PROGRAM PRG_ReadInputs
VAR
END_VAR

// -----------------------------------------------------------------------------
// OPERATOR CONTROLS
// -----------------------------------------------------------------------------
GVL_MASTER.stInputs.bStartButton                       := GVL_IO.stInputs.bStartButton;
GVL_MASTER.stInputs.bStopButton                        := GVL_IO.stInputs.bStopButton;
GVL_MASTER.stInputs.bResetButton                       := GVL_IO.stInputs.bResetButton;
GVL_MASTER.stInputs.bTwoHandsSafe                      := GVL_IO.stInputs.bTwoHandsSafe;

// -----------------------------------------------------------------------------
// PHYSICAL SAFETY DIAGNOSTICS
// -----------------------------------------------------------------------------
// These signals are used only to identify the physical cause of a safety drop.
// Machine Fault remains controlled by the validated TwinSAFE bSafetyOk signal.
GVL_MASTER.stInputs.bEmergencyStopChannel1             := GVL_IO.stInputs.bEmergencyStopChannel1;
GVL_MASTER.stInputs.bEmergencyStopChannel2             := GVL_IO.stInputs.bEmergencyStopChannel2;


// -----------------------------------------------------------------------------
// ELECTRICAL AND PROCESS DIAGNOSTICS
// -----------------------------------------------------------------------------
GVL_MASTER.stInputs.bUp24VPowerSupplyOk                 := GVL_IO.stInputs.bUp24VPowerSupplyOk;
GVL_MASTER.stInputs.bUs24VPowerSupplyOk                 := GVL_IO.stInputs.bUs24VPowerSupplyOk;
GVL_MASTER.stInputs.bIvekHeaterControllerAlarm          := GVL_IO.stInputs.bIvekHeaterControllerAlarm;
GVL_MASTER.stInputs.rIvekHeaterTemperature 				:= ((GVL_IO.stInputs.iIvekHeaterTemperature / 10.0) * (9.0 / 5.0)) + 32.0;
GVL_MASTER.stInputs.bSiliconeMinimumLevel1         		:= GVL_IO.stInputs.bSiliconeMinimumLevelSensor1;
GVL_MASTER.stInputs.bSiliconeMinimumLevel2         		:= GVL_IO.stInputs.bSiliconeMinimumLevelSensor2;


// -----------------------------------------------------------------------------
// DOOR AND PNEUMATIC DIAGNOSTICS
// -----------------------------------------------------------------------------
GVL_MASTER.stInputs.bMainDoorDiagnosticOk               := GVL_IO.stInputs.bMainDoorDiagnosticOk;
GVL_MASTER.stInputs.bMs6FeedbackOk                      := GVL_IO.stInputs.bMs6FeedbackOk;
GVL_MASTER.stInputs.bAirExhausted                       := GVL_IO.stInputs.bAirExhausted;

GVL_MASTER.stInputs.bMainDoorChannel1             		:= GVL_IO.stInputs.bMainDoorChannel1;
GVL_MASTER.stInputs.bMainDoorChannel2             		:= GVL_IO.stInputs.bMainDoorChannel2;
GVL_MASTER.stInputs.bMainDoorFeedback             		:= GVL_IO.stInputs.bMainDoorFeedback;

// -----------------------------------------------------------------------------
// FLAPS DIAGNOSTICS
// -----------------------------------------------------------------------------
GVL_MASTER.stInputs.bLeftFlapChannel1  					:= GVL_IO.stInputs.bLeftFlapChannel1;
GVL_MASTER.stInputs.bLeftFlapChannel2  					:= GVL_IO.stInputs.bLeftFlapChannel2;
GVL_MASTER.stInputs.bRightFlapChannel1 					:= GVL_IO.stInputs.bRightFlapChannel1;
GVL_MASTER.stInputs.bRightFlapChannel2 					:= GVL_IO.stInputs.bRightFlapChannel2;

// -----------------------------------------------------------------------------
// ANALOG PROCESS VALUES
// -----------------------------------------------------------------------------
// Raw terminal values are forwarded unchanged for diagnostics.
//
// Silicone and nozzle pressure sensors are connected to EL3064 voltage inputs.
// Commissioning measurements established a common zero around raw 3325 counts.
// The configured working scale is:
//     raw 3325  -> 0.00 bar
//     raw 16384 -> 10.00 bar
//
// This gives approximately:
//     Nozzle  raw 3910 -> 0.45 bar  (sensor display ~0.44 bar)
//     Silicone raw 5744 -> 1.85 bar (sensor display ~1.85 bar)
//
// Keep the raw values visible during commissioning so the scale can be refined
// later if a certified pressure reference is used.
GVL_MASTER.stInputs.uiMainAirPressureRaw               := GVL_IO.stInputs.uiMainAirPressureRaw;
GVL_MASTER.stInputs.uiSiliconePressureRaw              := GVL_IO.stInputs.uiSiliconePressureRaw;
GVL_MASTER.stInputs.uiNozzlePressureRaw                := GVL_IO.stInputs.uiNozzlePressureRaw;
GVL_MASTER.stInputs.uiVacuumPressureRaw                := GVL_IO.stInputs.uiVacuumPressureRaw;
GVL_MASTER.stInputs.uiExtractorFeedbackRaw 			   :=GVL_IO.stInputs.uiExtractionAVacuumPressureRaw;
GVL_MASTER.stInputs.iPartVacuumPressureRaw 				:= GVL_IO.stInputs.iPartVacuumPressureRaw;
// -----------------------------------------------------------------------------
// VACUUM EXTRACTOR FEEDBACK
// -----------------------------------------------------------------------------
// EL3064 Ch2.
// Approx. 250 = extractor OFF
// Approx. 700 = extractor ON


GVL_MASTER.stInputs.rSiliconePressureBar :=
    F_ScaleLinear(
        rRawValue := TO_REAL(GVL_IO.stInputs.uiSiliconePressureRaw),
        rRawMin   := GVL_Config.stMachine.stSiliconeSupply.rPressureRawLow,
        rRawMax   := GVL_Config.stMachine.stSiliconeSupply.rPressureRawHigh,
        rEngMin   := GVL_Config.stMachine.stSiliconeSupply.rSiliconePressureEngLow,
        rEngMax   := GVL_Config.stMachine.stSiliconeSupply.rSiliconePressureEngHigh
    );

GVL_MASTER.stInputs.rNozzlePressureBar :=
    F_ScaleLinear(
        rRawValue := TO_REAL(GVL_IO.stInputs.uiNozzlePressureRaw),
        rRawMin   := GVL_Config.stMachine.stSiliconeSupply.rPressureRawLow,
        rRawMax   := GVL_Config.stMachine.stSiliconeSupply.rPressureRawHigh,
        rEngMin   := GVL_Config.stMachine.stSiliconeSupply.rNozzlePressureEngLow,
        rEngMax   := GVL_Config.stMachine.stSiliconeSupply.rNozzlePressureEngHigh
    );

GVL_MASTER.stInputs.rVacuumEngineering :=
    F_ScaleLinear(
        rRawValue := TO_REAL(GVL_IO.stInputs.uiVacuumPressureRaw),
        rRawMin   := GVL_Config.stMachine.stSiliconeSupply.rVacuumRawLow,
        rRawMax   := GVL_Config.stMachine.stSiliconeSupply.rVacuumRawHigh,
        rEngMin   := GVL_Config.stMachine.stSiliconeSupply.rVacuumEngLow,
        rEngMax   := GVL_Config.stMachine.stSiliconeSupply.rVacuumEngHigh
    );


// Extractor running status with hysteresis.
IF NOT GVL_MASTER.stInputs.bExtractorRunning THEN

    IF GVL_MASTER.stInputs.uiExtractorFeedbackRaw >= 600 THEN
        GVL_MASTER.stInputs.bExtractorRunning := TRUE;
    END_IF

ELSE

    IF GVL_MASTER.stInputs.uiExtractorFeedbackRaw <= 400 THEN
        GVL_MASTER.stInputs.bExtractorRunning := FALSE;
    END_IF

END_IF

// Part holding vacuum feedback
IF NOT GVL_MASTER.stInputs.bPartVacuumOk THEN

    IF GVL_MASTER.stInputs.iPartVacuumPressureRaw >= 500 THEN
        GVL_MASTER.stInputs.bPartVacuumOk := TRUE;
    END_IF

ELSE

    IF GVL_MASTER.stInputs.iPartVacuumPressureRaw <= 400 THEN
        GVL_MASTER.stInputs.bPartVacuumOk := FALSE;
    END_IF

END_IF

// -----------------------------------------------------------------------------
// EVENT SYSTEM AGGREGATES
// -----------------------------------------------------------------------------
// These values are generated by the event manager and consumed by the machine
// state logic. Individual diagnostic conditions remain inside PRG_Events.
GVL_MASTER.stInputs.bEventFault                        := GVL_MASTER.bMachineFault;
GVL_MASTER.stInputs.bEventCycleStopRequest             := GVL_MASTER.bCycleStopRequest;

// -----------------------------------------------------------------------------
// SAFETY INTERFACE
// -----------------------------------------------------------------------------
// bSafetyOk is the validated TwinSAFE aggregate used by the machine state logic.
// Individual physical safety signals are used separately for diagnostics.
GVL_MASTER.stInputs.stSafety.bSafetyOk                 := GVL_IO.stInputs.bSafetyOk;

// Safety-only permissions. Operational conditions such as part presence,
// cylinder positions and process readiness belong to the machine permissives.
GVL_MASTER.stInputs.stSafety.bMotionSafetyPermitted    := GVL_IO.stInputs.bSafetyOk;
GVL_MASTER.stInputs.stSafety.bProcessSafetyPermitted   := GVL_MASTER.stInputs.stSafety.bMotionSafetyPermitted;

// -----------------------------------------------------------------------------
// PART DETECTION
// -----------------------------------------------------------------------------
GVL_MASTER.stInputs.bGearboxAssemblyPartPresent        := GVL_IO.stInputs.bGearboxAssemblyPartPresent;
GVL_MASTER.stInputs.bReservoirPartPresent              := GVL_IO.stInputs.bReservoirPartPresent;
GVL_MASTER.stInputs.bBothPartPresent                   := GVL_IO.stInputs.bBothPartPresent;
GVL_MASTER.stInputs.bRejectChutePartPresent            := GVL_IO.stInputs.bRejectChutePartPresent;
GVL_MASTER.stInputs.bSiliconeStationPartPresent 	    :=GVL_IO.stInputs.bSiliconeStationPartPresent;

// -----------------------------------------------------------------------------
// INDEX TABLE
// -----------------------------------------------------------------------------
GVL_MASTER.stInputs.bIndexReady                        := GVL_IO.stInputs.bIndexReady;
GVL_MASTER.stInputs.bIndexLocked                       := GVL_IO.stInputs.bIndexLocked;
GVL_MASTER.stInputs.bIndexCompletedSensor              := GVL_IO.stInputs.bIndexCompletedSensor;
GVL_MASTER.stInputs.bIndexSupportExtended              := GVL_IO.stInputs.bIndexSupportExtended;
GVL_MASTER.stInputs.bIndexSupportRetracted             := GVL_IO.stInputs.bIndexSupportRetracted;
GVL_MASTER.stInputs.eIndexPosition                     := GVL_IO.stInputs.eIndexPosition;

// -----------------------------------------------------------------------------
// MAIN DOOR
// -----------------------------------------------------------------------------
GVL_MASTER.stInputs.bMainDoorClosed                    := GVL_IO.stInputs.bMainDoorClosed;
GVL_MASTER.stInputs.bMainDoorLocked                    := GVL_IO.stInputs.bMainDoorLocked;
GVL_MASTER.stInputs.bMainDoorUnsafe                    := GVL_IO.stInputs.bMainDoorUnsafe;

// -----------------------------------------------------------------------------
// PROCESS SUPPORT CYLINDERS
// -----------------------------------------------------------------------------
// Electrical drawing: Transfer Nest Support.
// Software terminology: Silicone Support.
GVL_MASTER.stInputs.bSiliconeSupportExtended           := GVL_IO.stInputs.bSiliconeSupportExtended;
GVL_MASTER.stInputs.bSiliconeSupportRetracted          := GVL_IO.stInputs.bSiliconeSupportRetracted;
GVL_MASTER.stInputs.bAssemblySupportExtended           := GVL_IO.stInputs.bAssemblySupportExtended;
GVL_MASTER.stInputs.bAssemblySupportRetracted          := GVL_IO.stInputs.bAssemblySupportRetracted;

// Flipping / assembly station
GVL_MASTER.stInputs.bTransferVerticalMiniSlideRetracted := GVL_IO.stInputs.bTransferVerticalMiniSlideRetracted;
GVL_MASTER.stInputs.bTransferVerticalMiniSlideExtended  := GVL_IO.stInputs.bTransferVerticalMiniSlideExtended;
GVL_MASTER.stInputs.bRotaryGripperOpened                := GVL_IO.stInputs.bRotaryGripperOpened;
GVL_MASTER.stInputs.bRotaryGripperClosed                := GVL_IO.stInputs.bRotaryGripperClosed;
GVL_MASTER.stInputs.bRotaryGripperRotationPick0         := GVL_IO.stInputs.bRotaryGripperRotationPick0;
GVL_MASTER.stInputs.bRotaryGripperRotationPlace180      := GVL_IO.stInputs.bRotaryGripperRotationPlace180;


// -----------------------------------------------------------------------------
// IVEK ETHERNET/IP INTERFACE
// -----------------------------------------------------------------------------
GVL_IVEK_EIP.bCommunicationOk 						   := (GVL_IVEK_EIP.stInput.usiIvekConnectionState = 0);
GVL_MASTER.stIvekInput                                 := GVL_IVEK_EIP.stInput;
GVL_MASTER.bIvekCommsOk                                := GVL_IVEK_EIP.bCommunicationOk;

END_PROGRAM

(* stored: Version 1.1.0.1, ProductVersion 3.1.4026.18
   POU PRG_ReadInputs: Id {743776ea-f060-4d26-80b1-ea31dbcde434}, SpecialFunc None *)
